INTERFACE IFileData_t

METHOD getDataPtr : POINTER TO BYTE
END_METHOD

METHOD getSize : UDINT
VAR_INPUT
END_VAR
END_METHOD

END_INTERFACE

(* stored: Version 1.1.0.1, ProductVersion 3.1.4024.13
   Itf IFileData_t: Id {d3a5a00e-a1d7-415f-9d71-ec953fc53d9c}
   Method getDataPtr: Id {8ee49171-46d8-42d1-aff3-8925c0b66377}
   Method getSize: Id {191272b1-c804-462b-bc3e-038ca6fa97ef} *)
